// TIA Portal V18 export
VAR_GLOBAL   // PLC tag table "Alert"
   iBEmerencia AT %I16.2 : Bool;
   oSirene AT %Q17.1 : Bool;
END_VAR
